// TIA Portal V17 export
// export: Created 2022-07-20T07:02:40.3993455Z, ExportSetting WithDefaults, DisplayName Totally Integrated Automation Portal, DisplayVersion V17, DisplayName TIA Portal Openness, DisplayVersion V17, DisplayName TIA Portal Version Control Interface, DisplayVersion V17, DisplayName SINAMICS Startdrive Advanced, DisplayVersion V17, DisplayName SINAMICS Startdrive G130, G150, S120, S150, SINAMICS MV, S210, DisplayVersion V17, DisplayName SINAMICS Startdrive G110M, G120, G120C, G120D, G120P, G115D, DisplayVersion V17, DisplayName STEP 7 Professional, DisplayVersion V17, DisplayName STEP 7 Safety, DisplayVersion V17, DisplayName WinCC Advanced, DisplayVersion V17
VAR_GLOBAL   // PLC tag table "LCon_ExampleTags"
END_VAR
VAR_GLOBAL CONSTANT   // user constants
   WINDER_BOTTOM : Int := 2;
   NUMBER_OF_WINDER : Int := 3;   // Number of winders: 1 - x
   NUMBER_OF_SECTIONAL_DRIVES : Int := 2;   // Number of sectional drives 1 - x
   "0_WINDER_STATE_IDLE" : Int := 0;
   "10_WINDER_STATE_ENABLE_AXIS" : Int := 10;
   "20_WINDER_STATE_WAIT_AXIS_ENABLED" : Int := 20;
   "30_WINDER_STATE_AXIS_ENABLED" : Int := 30;
   "40_WINDER_STATE_ENABLE_FB" : Int := 40;
   "50_WINDER_STATE_WAIT_FB_ENABLED" : Int := 50;
   "70_WINDER_STATE_ENABLE_CONTROL" : Int := 70;
   "80_WINDER_STATE_WAIT_CONTROL_ENABLED" : Int := 80;
   "90_WINDER_STATE_WINDER_IN_OPERATION" : Int := 90;
   "200_WINDER_STATE_DISABLE_CONTROL" : Int := 200;
   "210_WINDER_STATE_WAIT_CONTROL_DISABLED" : Int := 210;
   "220_WINDER_STATE_CONTROL_DISABLED" : Int := 220;
   "230_WINDER_STATE_DISABLE_FB" : Int := 230;
   "240_WINDER_STATE_WAIT_FB_DISABLED" : Int := 240;
   "250_WINDER_STATE_FB_DISABLED" : Int := 250;
   "260_WINDER_STATE_DISABLE_AXIS" : Int := 260;
   "270_WINDER_STATE_WAIT_AXIS_DISABLED" : Int := 270;
   "900_WINDER_STATE_ERROR" : Int := 900;
   "0_MAIN_STATE_IDLE" : Int := 0;
   "10_MAIN_STATE_ENABLE_INFEED_MASTER" : Int := 10;
   "20_MAIN_STATE_WAIT_INFEED_MASTER_ENABLED" : Int := 20;
   "30_MAIN_STATE_INFEED_MASTER_ENABLED" : Int := 30;
   "70_MAIN_STATE_ENABLE_MODULES" : Int := 70;
   "80_MAIN_STATE_WAIT_MODULES_ENABLED" : Int := 80;
   "90_MAIN_STATE_MODULES_READY_TO_START" : Int := 90;
   "100_MAIN_STATE_MODULES_IN_OPERATION" : Int := 100;
   "110_MAIN_STATE_DISABLE_MODULES" : Int := 110;
   "120_MAIN_STATE_WAIT_MODULES_DISABLED" : Int := 120;
   "160_MAIN_STATE_DISABLE_INFEED_MASTER" : Int := 160;
   "900_MAIN_STATE_ERROR" : Int := 900;
   "0_LINE_STATE_IDLE" : Int := 0;
   "10_LINE_STATE_ENABLE_FB" : Int := 10;
   "20_LINE_STATE_WAIT_FB_ENABLED" : Int := 20;
   "30_LINE_STATE_FB_ENABLED" : Int := 30;
   "40_LINE_STATE_ENABLE_AXIS" : Int := 40;
   "50_LINE_STATE_WAIT_AXIS_ENABLED" : Int := 50;
   "100_LINE_STATE_READY_TO_START" : Int := 100;
   "110_LINE_STATE_START_LINE" : Int := 110;
   "120_LINE_STATE_LINE_IN_MOTION" : Int := 120;
   "130_LINE_STATE_STOP_LINE" : Int := 130;
   "140_LINE_STATE_LINE_STOPPING" : Int := 140;
   "150_LINE_STATE_LINE_STOPPED" : Int := 150;
   "220_LINE_STATE_DISABLE_AXIS" : Int := 220;
   "230_LINE_STATE_WAIT_AXIS_DISABLED" : Int := 230;
   "240_LINE_STATE_DISABLE_FB" : Int := 240;
   "250_LINE_STATE_WAIT_FB_DISABLED" : Int := 250;
   "260_LINE_STATE_FB_DISABLED" : Int := 260;
   "900_LINE_STATE_ERROR" : Int := 900;
   "0_SECTIONAL_STATE_IDLE" : Int := 0;
   "10_SECTIONAL_STATE_ENABLE_AXIS" : Int := 10;
   "20_SECTIONAL_STATE_WAIT_AXIS_ENABLED" : Int := 20;
   "30_SECTIONAL_STATE_AXIS_ENABLED" : Int := 30;
   "40_SECTIONAL_STATE_ENABLE_FB" : Int := 40;
   "50_SECTIONAL_STATE_WAIT_FB_ENABLED" : Int := 50;
   "60_SECTIONAL_STATE_FB_ENABLED" : Int := 60;
   "70_SECTIONAL_STATE_ENABLE_CONTROL" : Int := 70;
   "80_SECTIONAL_STATE_WAIT_CONTROL_ENABLED" : Int := 80;
   "90_SECTIONAL_STATE_IN_OPERATION" : Int := 90;
   "200_SECTIONAL_STATE_DISABLE_CONTROL" : Int := 200;
   "210_SECTIONAL_STATE_WAIT_CONTROL_DISABLED" : Int := 210;
   "220_SECTIONAL_STATE_CONTROL_DISABLED" : Int := 220;
   "230_SECTIONAL_STATE_DISABLE_FB" : Int := 230;
   "240_SECTIONAL_STATE_WAIT_FB_DISABLED" : Int := 240;
   "250_SECTIONAL_STATE_FB_DISABLED" : Int := 250;
   "260_SECTIONAL_STATE_DISABLE_AXIS" : Int := 260;
   "270_SECTIONAL_STATE_WAIT_AXIS_DISABLED" : Int := 270;
   "900_SECTIONAL_STATE_ERROR" : Int := 900;
   UNWINDER_AXIS : Int := 1;
   "160_LINE_STATE_POS_LINE_FW" : Int := 160;
   "180_LINE_STATE_IN_POSITION_FW" : Int := 180;
   "170_LINE_STATE_POSITIONING_FW" : Int := 170;
   "190_LINE_STATE_POS_LINE_REV" : Int := 190;
   "40_MAIN_STATE_ENABLE_BUFFER" : Int := 40;
   "50_MAIN_STATE_WAIT_BUFFER_ENABLED" : Int := 50;
   "60_MAIN_STATE_BUFFER_ENABLED" : Int := 60;
   "130_MAIN_STATE_DISABLE_BUFFER" : Int := 130;
   "140_MAIN_STATE_WAIT_BUFFER_DISABLED" : Int := 140;
   "150_MAIN_STATE_BUFFER_DISABLED" : Int := 150;
   "180_MAIN_STATE_INFEED_MASTER_DISABLED" : Int := 180;
   "170_MAIN_STATE_WAIT_INFEED_MASTER_DISABLED" : Int := 170;
   "60_LINE_STATE_HOME_AXIS" : Int := 60;
   "70_LINE_STATE_WAIT_AXIS_HOMED" : Int := 70;
   "80_LINE_STATE_GEARIN_SLAVE_AXIS" : Int := 80;
END_VAR
